FUNCTION_BLOCK FB_SimpleLinearTwoWayDrive
VAR_INPUT
	SensorHomePos: BOOL;
	SensorWorkPos: BOOL;
	Enable: BOOL;
	ToHome: BOOL;
	ToWork: BOOL;
END_VAR
VAR_OUTPUT
	ActorHomePos: BOOL;
	ActorWorkPos: BOOL;
END_VAR
VAR
END_VAR

ActorHomePos := Enable AND ToHome AND NOT ActorWorkPos AND NOT SensorHomePos;
ActorWorkPos := Enable AND ToWork AND NOT ActorHomePos AND NOT SensorWorkPos;

END_FUNCTION_BLOCK

(* stored: Version 1.1.0.1, ProductVersion 3.1.4024.11
   POU FB_SimpleLinearTwoWayDrive: Id {d5079cf3-2029-4674-b5d0-714b53c5075a}, SpecialFunc None *)
